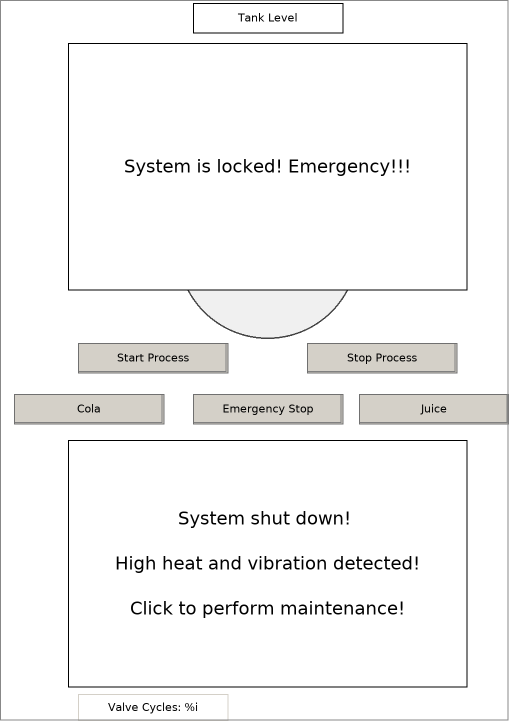
VISUALIZATION Visualization  // 509x721
    BarDisplayImage (119,43 300x50), value: GVL_Process.fCurrentLevel, style: BarDisplayImage-Gray, scale format: %.1f, scale 0..1000
    Meter360 (177,150 181x196), value: GVL_Process.fCurrentTemp, style: Meter-Meter360-Gray, scale format: %.1f, scale 0..100
    Rectangle (193,3 150x30), "Tank Level"
    Rectangle (193,103 150x30), "Temperature"
    Button (78,343 150x30), "Start Process"
        OnMouseClick: execute { GVL_Process.bStartProcess := TRUE; }
    Button (193,394 150x30), "Emergency Stop"
        toggle GVL_Process.bEmergencyStop
    Button (14,394 150x30), "Cola"
        tap GVL_Process.bColaActive
        OnMouseClick: execute { GVL_Process.nSelectedRecipe := 1; }
    Button (359,394 150x30), "Juice"
        tap GVL_Process.bJuiceActive
        OnMouseClick: execute { GVL_Process.nSelectedRecipe := 2; }
    Rectangle (102,520 78x18), "VALF"
    Rectangle (233,520 78x18), "HEATING"
    Rectangle (359,520 78x18), "MIXER"
    Lamp1 (110,440 70x70), variable: GVL_Process.bInletValve, style: Lamp-Lamp1-Yellow
    Lamp1 (241,440 70x70), variable: GVL_Process.bHeater, style: Lamp-Lamp1-Yellow
    Lamp1 (359,440 70x70), variable: GVL_Process.bMixerMotor, style: Lamp-Lamp1-Yellow
    Textfield (78,599 150x30), "Total Bottles Produced: %i", text variable: GVL_Process.nTotalBottles
    Rectangle (68,43 399x247), "System is locked! Emergency!!!", invisible if: NOT GVL_Process.bEmergencyStop
    Textfield (78,554 372x28), "Status: %s", text variable: GVL_Process.sStatusMessage
    Button (307,343 150x30), "Stop Process"
        OnMouseClick: execute { GVL_Process.bStartProcess := FALSE; }
    Textfield (279,599 150x30), "Cola Produced: %i", text variable: GVL_Process.nColaCount
    Textfield (78,644 150x30), "Now Producing: %s", text variable: GVL_Process.sCurrentProduct
    Textfield (279,644 150x30), "Juice Produced: %i", text variable: GVL_Process.nJuiceCount
    Textfield (78,694 150x27), "Valve Cycles: %i", text variable: GVL_Process.nValveCycleCount
    Rectangle (68,440 399x247), "System shut down! High heat and vibration detected! Click to perform maintenance!", invisible if: NOT GVL_Process.bMaintenanceAlarm
        OnMouseClick: execute { GVL_Process.bMaintenanceAlarm := FALSE; }
END_VISUALIZATION

(* stored: Version 1.1.0.1
   Visu Visualization: Id {3541133c-bbf2-4103-8958-df6fbbc8a96a} *)
